{attribute addProperty BoxType "EL2624-0000-0016"}
{attribute addProperty Id "ChannelAT %Q*ARRAY[0..3] OF Channel_7F374EB03240WcStateAT %I*WcState_28A8677510.1250InfoDataAT %I*InfoData_192954DE1620"}
{attribute addProperty CRC "2753798610"}
{attribute addProperty SizeInBites "49"}
{attribute addProperty SizeInBytes "6.125"}
TYPE EL2624_4E3C7537 :
STRUCT
	{attribute addProperty Name "Channel"}
	Channel : ARRAY[0..3] OF Channel_7F374EB0;
	{attribute addProperty Name "WcState"}
	WcState : WcState_28A86775;
	{attribute addProperty Name "InfoData"}
	InfoData : InfoData_192954DE;
END_STRUCT
END_TYPE

(* stored: Version 1.2.0.0, ProductVersion 3.1.4024.9
   DUT EL2624_4E3C7537: Id {4247a1f9-fa4b-4d59-8c6a-18fdde3ce1ef} *)
